(****************************************************************
NAME:			FB_CoupleAxis
DATA:			2017.2.16
VERSION:		1.0.0
DESCRIPTION:	FB_CoupleAxis
HISTORY:
				2017.2.16		NEW

***************************************************************)
FUNCTION_BLOCK FB_CoupleAxis
VAR_INPUT
	Execute:BOOL;
	Reset:BOOL;
END_VAR
VAR_OUTPUT
	FbID:DINT:=1001;
	State:DINT;
	Busy:BOOL;
	InGear:BOOL;
	Error:BOOL;
	ErrorID:DINT;
END_VAR
VAR_IN_OUT
END_VAR
VAR
	Bottom_MC_GearIn: MC_GearIn;
	Top_MC_GearIn: MC_GearIn;
	fb_ton: TON;
END_VAR

IF Execute THEN
Busy:=TRUE;
InGear:=FALSE;
fb_ton(PT:=t#0.1s);
CASE State OF
	0:	(*Check*)
		IF LeftTopLin.NcToPlc.CoupleState=3 OR LeftBottomLin.NcToPlc.CoupleState=3 THEN	(*LeftTop»òÕßLeftBottomÎª´ÓÖá£¬Emergency Error*)
			ErrorID:=1;
			State:=-100;
		ELSIF LeftTopLin.NcToPlc.CoupleState=2 OR LeftBottomLin.NcToPlc.CoupleState=2
			OR RightTopLin.NcToPlc.CoupleState=2 OR RightBottomLin.NcToPlc.CoupleState=2 THEN	(*ÓÐÒ»ÖáCoupleStateÎª2£¬Emergency Error*)
			ErrorID:=2;
			State:=-100;
		ELSIF LeftTopLin.NcToPlc.CoupleState=1 AND LeftBottomLin.NcToPlc.CoupleState=1
			AND RightTopLin.NcToPlc.CoupleState=3 AND RightBottomLin.NcToPlc.CoupleState=3 THEN	(*ÒÑ¾­´¦ÓÚñîºÏ×´Ì¬*)
			ErrorID:=3;
			State:=-100;
		ELSIF LeftTopLin.Status.Moving OR  RightTopLin.Status.Moving OR LeftBottomLin.Status.Moving OR RightBottomLin.Status.Moving THEN	(*ÓÐÖáÔË¶¯*)
			ErrorID:=4;
			State:=-100;
		ELSIF  Top_MC_GearIn.Error OR Bottom_MC_GearIn.Error THEN		(*FB Error*)
			ErrorID:=5;
			State:=99;
		ELSIF Top_MC_GearIn.InGear OR Bottom_MC_GearIn.InGear THEN	(*ÒÑ¾­InGear£¬²»¿ÉÄÜ·¢Éú£¬FB Error*)
			ErrorID:=6;
			State:=99;
		ELSIF LeftTopLin.NcToPlc.CoupleState=0 AND LeftBottomLin.NcToPlc.CoupleState=0
			AND RightTopLin.NcToPlc.CoupleState=0 AND RightBottomLin.NcToPlc.CoupleState=0 THEN	(*Öá¾ù´¦ÓÚÎÞñîºÏ×´Ì¬£¬×ªÏÂÒ»²½*)
			State:=1;
		ELSE
			ErrorID:=7;
			State:=-100;
		END_IF
	1:	(*Couple*)
		IF LeftTopLin.NcToPlc.CoupleState=0 AND LeftBottomLin.NcToPlc.CoupleState=0
			AND RightTopLin.NcToPlc.CoupleState=0 AND RightBottomLin.NcToPlc.CoupleState=0 THEN	(*ÔÙ¼ì²é£¬Öá¾ù´¦ÓÚÎÞñîºÏ×´Ì¬£¬¿ªÊ¼ñîºÏ*)
			Top_MC_GearIn.Execute:=TRUE;
			Bottom_MC_GearIn.Execute:=TRUE;
			A_CoupleMC();
			fb_ton.IN:=TRUE;
			State:=2;
		ELSE
			ErrorID:=7;
			State:=99;
		END_IF
	2:	(*Couple Wait*)
		A_CoupleMC();
		IF NOT Top_MC_GearIn.InGear OR NOT Bottom_MC_GearIn.InGear THEN		(*InGearÐÅºÅ²»µ½£¬¼ÌÐøµÈ´ý£¬Èç¹û³¬Ê±ÔòFB Error*)
			IF NOT fb_ton.Q THEN
				State:=2;
			ELSE
				ErrorID:=8;
				State:=99;
			END_IF
		ELSIF  LeftTopLin.NcToPlc.CoupleState<>1 OR  RightTopLin.NcToPlc.CoupleState<>3
			OR LeftBottomLin.NcToPlc.CoupleState<>1 OR  RightBottomLin.NcToPlc.CoupleState<>3 THEN		(*ñîºÏ×´Ì¬²»¶Ô£¬Emergency Error*)
				ErrorID:=9;
				State:=-100;
		ELSIF   LeftTopLin.NcToPlc.CoupleState=1 AND  RightTopLin.NcToPlc.CoupleState=3
			AND LeftBottomLin.NcToPlc.CoupleState=1 AND  RightBottomLin.NcToPlc.CoupleState=3 THEN		(*ÕýÈ·ñîºÏ×´Ì¬£¬×ªÏÂÒ»²½*)
				State:=88;
		ELSE
				ErrorID:=10;
				State:=-100;
		END_IF
	88:	(*InGear*)
		Execute:=FALSE;
		State:=0;
		Busy:=FALSE;
		InGear:=TRUE;
		Error:=FALSE;
		ErrorID:=0;
		Bottom_MC_GearIn.Execute:=FALSE;
		Top_MC_GearIn.Execute:=FALSE;
		A_CoupleMC();
		fb_ton.IN:=FALSE;
	99:	(*FB Error*)
		Execute:=FALSE;
		State:=99;
		Busy:=FALSE;
		InGear:=FALSE;
		Error:=TRUE;
		Bottom_MC_GearIn.Execute:=FALSE;
		Top_MC_GearIn.Execute:=FALSE;
		A_CoupleMC();
		fb_ton.IN:=FALSE;
	-100:	(*Emergency Error*)
		FB_PlcEmergencyStop();
		Execute:=FALSE;
		State:=-100;
		Busy:=FALSE;
		InGear:=FALSE;
		Error:=TRUE;
		Bottom_MC_GearIn.Execute:=FALSE;
		Top_MC_GearIn.Execute:=FALSE;
		A_CoupleMC();
		fb_ton.IN:=FALSE;
END_CASE
END_IF
IF Reset THEN
		Execute:=FALSE;
		State:=0;
		Busy:=FALSE;
		InGear:=FALSE;
		Error:=FALSE;
		ErrorID:=0;
		Bottom_MC_GearIn.Execute:=FALSE;
		Top_MC_GearIn.Execute:=FALSE;
		A_CoupleMC();
		Reset:=FALSE;
END_IF

ACTION A_CoupleMC:
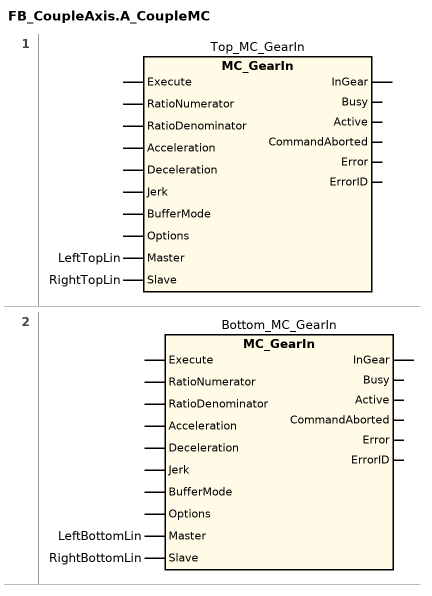
// NETWORK 1
Top_MC_GearIn(Master := LeftTopLin, Slave := RightTopLin); // MC_GearIn

// NETWORK 2
Bottom_MC_GearIn(Master := LeftBottomLin, Slave := RightBottomLin); // MC_GearIn
END_ACTION

END_FUNCTION_BLOCK

(* stored: Version 1.1.0.1, ProductVersion 3.1.4024.6
   POU FB_CoupleAxis: Id {e9d1561f-4b1b-4266-afdb-4fc5f4697c02}, SpecialFunc None
   Action A_CoupleMC: Id {392f47cf-c823-4531-a98e-b3b71519aae7} *)
